FUNCTION_BLOCK FB_SendVelocityGains_Right
VAR_INPUT
	ProportionalGain : LREAL;
	IntegralGain : LREAL;
	InitialIntegralValue : LREAL;
END_VAR
VAR_OUTPUT
END_VAR
VAR
	TxMessage : EXTCANQUEUE;
	i : INT;
	ProportionalGain_Values : ARRAY[0..1] OF BYTE;
	IntegrallGain_Values : ARRAY[0..1] OF BYTE;
	InitialIntegralValue_Values : ARRAY[0..3] OF BYTE;
END_VAR
VAR_IN_OUT
	CAN_OUTPUTS_Right : CANTXQUEUESTRUCT_E_32;
	CAN_INPUTS_Right : CANRXQUEUESTRUCT_E_32;
END_VAR

(*ProportionalGain_Values[1] := DINT_TO_BYTE(LREAL_TO_DINT(ProportionalGain*100) AND 16#FF);
ProportionalGain_Values[0] := DINT_TO_BYTE(SHR(LREAL_TO_DINT(ProportionalGain*100), 8) AND 16#FF);

IntegrallGain_Values[1] := DINT_TO_BYTE(LREAL_TO_DINT(IntegralGain*100) AND 16#FF);
IntegrallGain_Values[0] := DINT_TO_BYTE(SHR(LREAL_TO_DINT(IntegralGain*100), 8) AND 16#FF);

InitialIntegralValue_Values[1] := DINT_TO_BYTE(LREAL_TO_DINT(InitialIntegralValue*100) AND 16#FF);
InitialIntegralValue_Values[0] := DINT_TO_BYTE(SHR(LREAL_TO_DINT(InitialIntegralValue*100), 8) AND 16#FF);*)

ProportionalGain_Values[1] := DINT_TO_BYTE(LREAL_TO_DINT(ProportionalGain*1) AND 16#FF);
ProportionalGain_Values[0] := DINT_TO_BYTE(SHR(LREAL_TO_DINT(ProportionalGain*1), 8) AND 16#FF);

IntegrallGain_Values[1] := DINT_TO_BYTE(LREAL_TO_DINT(IntegralGain*1) AND 16#FF);
IntegrallGain_Values[0] := DINT_TO_BYTE(SHR(LREAL_TO_DINT(IntegralGain*1), 8) AND 16#FF);

InitialIntegralValue_Values[3] := DINT_TO_BYTE(LREAL_TO_DINT(InitialIntegralValue*100) AND 16#FF);
InitialIntegralValue_Values[2] := DINT_TO_BYTE(SHR(LREAL_TO_DINT(InitialIntegralValue*100), 8) AND 16#FF);
InitialIntegralValue_Values[1] := DINT_TO_BYTE(SHR(LREAL_TO_DINT(InitialIntegralValue*100), 16) AND 16#FF);
InitialIntegralValue_Values[0] := DINT_TO_BYTE(SHR(LREAL_TO_DINT(InitialIntegralValue*100), 24) AND 16#FF);

TxMessage.cobId := 310;
TxMessage.length := 8;
FOR i := 0 TO 7 DO 
	IF i < 2 THEN 
		TxMessage.data[i] := ProportionalGain_Values[i];
	ELSIF i < 4 THEN
		TxMessage.data[i] := IntegrallGain_Values[i - 2];
	ELSE 
		TxMessage.data[i] := InitialIntegralValue_Values[i - 4];
	END_IF
END_FOR
CAN_OUTPUTS_Right.TxMessages[7] := TxMessage;
//CAN_OUTPUTS.NoOfTxMessages := 1

END_FUNCTION_BLOCK

(* stored: Version 1.1.0.1
   POU FB_SendVelocityGains_Right: Id {9614ac6a-ae01-4b85-a328-a66f7418117f}, SpecialFunc None *)
